Omron CX-Programmer project NewProject (CX-Programmer 9.73)

# PLC NewPLC1: CP1E N30

## Program NewProgram1 (cyclic task 0)

### Section Section1

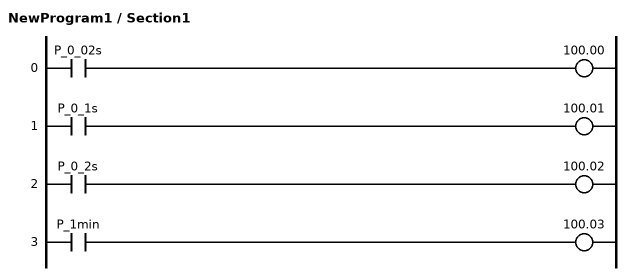
; rung 0
LD P_0_02s
OUT 100.00
; rung 1
LD P_0_1s
OUT 100.01
; rung 2
LD P_0_2s
OUT 100.02
; rung 3
LD P_1min
OUT 100.03

### Section END
; rung 0
END(001)